// TIA Portal V21 export
ORGANIZATION_BLOCK "Startup"   // OB100, LAD, Startup
TITLE = "Complete Restart"
{ S7_Optimized_Access := 'TRUE' }
// stored: SetENOAutomatically false
   VAR_INPUT
      LostRetentive : Bool;   // True if retentive data are lost
      LostRTC : Bool;   // True if date and time are lost
   END_VAR
BEGIN

REGION Network 1 (SCL): Load the selected hardware combination
   // The configuration of the slots is loaded according to the selected hardware combination
   IF (("C0_ID".CabinetNumber >= 1) AND ("C0_ID".CabinetNumber <= "K_MaxCabinetNumber")) THEN
       "HWData".CombiNumber := "Cabinets_Config".C0["C0_ID".CabinetNumber].HWCombiNumber;
       IF (("HWData".CombiNumber >= 1) AND ("HWData".CombiNumber <= "K_MaxHWCombiNumber")) THEN
           "HWData".CPUET200SP_Config := "HWData".ConfigSlots["HWData".CombiNumber];
           "C0_DATA".C0 := "Cabinets_Config".C0["C0_ID".CabinetNumber];
       ELSE
           "M_HWCombiNumberOutOfRange" := TRUE;
       END_IF;
   ELSE
       "M_CabinetNumberOutOfRange" := TRUE;
   END_IF;
END_REGION

REGION Network 2: Hardware configuration
   // For more details refer to:
   // - Configuring standard machines in TIA Portal (configuration control) Application example.
   // - Library for Configuration Control (LCC).
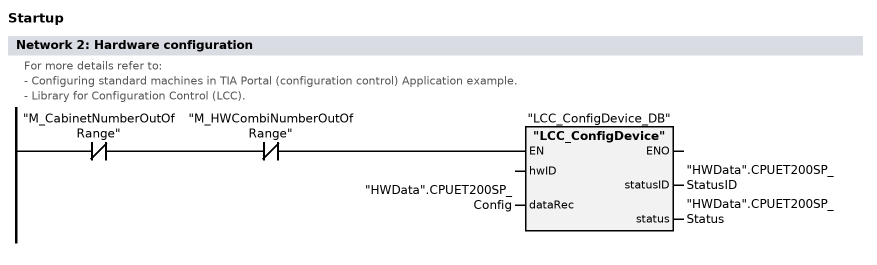
   RUNG wire#powerrail
      I_Contact( "M_CabinetNumberOutOfRange" )
      I_Contact( "M_HWCombiNumberOutOfRange" )
      "LCC_ConfigDevice_DB"(hwID :=, dataRec := "HWData".CPUET200SP_Config, statusID => "HWData".CPUET200SP_StatusID, status => "HWData".CPUET200SP_Status)
   END_RUNG
   // the same network as SCL:
   IF NOT "M_CabinetNumberOutOfRange" AND NOT "M_HWCombiNumberOutOfRange" THEN
       "LCC_ConfigDevice_DB"(dataRec := "HWData".CPUET200SP_Config,   // "LCC_ConfigDevice"
                             statusID => "HWData".CPUET200SP_StatusID,
                             status => "HWData".CPUET200SP_Status);
   END_IF;
END_REGION

REGION Network 3 (SCL): Configuration of the +C0 cabinet functionalities according to the configured hardware.
   // For all hardware combinations:
   //   - Power lines L1/L2 are always available.
   //   - Safety zones Z1/Z2 are always available.
   IF "HWData".CombiNumber > 4 THEN
       "M_Power_line_3_4_Available" := TRUE;
       "M_Safety_zone_3_4_Available" := TRUE;
   END_IF;

   IF "HWData".CombiNumber > 8 THEN
       "M_Power_line_5_6_Available" := TRUE;
       "M_Safety_zone_5_6_Available" := TRUE;
   END_IF;

   IF "HWData".CombiNumber > 12 THEN
       "M_Safety_zone_7_8_Available" := TRUE;
   END_IF;

   IF ("HWData".CombiNumber = 2 OR
       "HWData".CombiNumber = 6 OR
       "HWData".CombiNumber = 10 OR
       "HWData".CombiNumber = 14) THEN
       "M_Wrapping_machine_Enabled" := TRUE;
   END_IF;

   IF ("HWData".CombiNumber = 3 OR
       "HWData".CombiNumber = 7 OR
       "HWData".CombiNumber = 11 OR
       "HWData".CombiNumber = 15) THEN
       "M_Fast_doors_Enabled" := TRUE;
   END_IF;

   IF ("HWData".CombiNumber = 4 OR
       "HWData".CombiNumber = 8 OR
       "HWData".CombiNumber = 12 OR
       "HWData".CombiNumber = 16) THEN
       "M_Wrapping_machine_Enabled" := TRUE;
       "M_Fast_doors_Enabled" := TRUE;
   END_IF;
END_REGION
END_ORGANIZATION_BLOCK
